% RSLogix 500 project LAB3_BW_OJ_BAK001.RSS, saved by version 8.40.00.08 %
PROJECT "UNTITLED"    % processor: MicroLogix 1400 %

PROGRAM FILES
  LAD 2   6 rungs

DATA FILES
  O0 OUTPUT  6 elements
  I1 INPUT  8 elements
  S2 STATUS  66 elements
  B3 BINARY  1 elements
  T4 TIMER  1 elements
  C5 COUNTER  1 elements
  R6 CONTROL  1 elements
  N7 INTEGER  1 elements
  F8 FLOAT  1 elements

LADDER 2
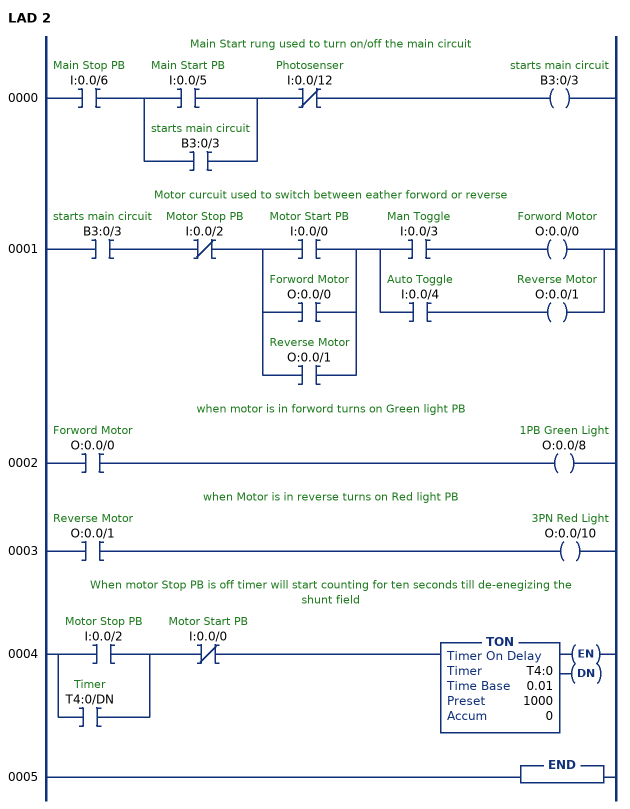
% Rung: 0 %
% Main Start rung used to turn on/off the main circuit %
SOR XIC I:0.0/6 BST XIC I:0.0/5 NXB XIC B3:0/3 BND XIO I:0.0/12 OTE B3:0/3 EOR
%   I:0.0/6  "Main Stop PB" %
%   I:0.0/5  "Main Start PB" %
%   B3:0/3  "starts main circuit" %
%   I:0.0/12  "Photosenser" %
% Rung: 1 %
% Motor curcuit used to switch between eather forword or reverse %
SOR XIC B3:0/3 XIO I:0.0/2 BST XIC I:0.0/0 NXB XIC O:0.0/0 NXB XIC O:0.0/1 BND BST XIC I:0.0/3 OTE O:0.0/0 NXB XIC I:0.0/4 OTE O:0.0/1 BND EOR
%   B3:0/3  "starts main circuit" %
%   I:0.0/2  "Motor Stop PB" %
%   I:0.0/0  "Motor Start PB" %
%   O:0.0/0  "Forword Motor" %
%   O:0.0/1  "Reverse Motor" %
%   I:0.0/3  "Man Toggle" %
%   I:0.0/4  "Auto Toggle" %
% Rung: 2 %
% when motor is in forword turns on Green light PB %
SOR XIC O:0.0/0 OTE O:0.0/8 EOR
%   O:0.0/0  "Forword Motor" %
%   O:0.0/8  "1PB Green Light" %
% Rung: 3 %
% when Motor is in reverse turns on Red light PB %
SOR XIC O:0.0/1 OTE O:0.0/10 EOR
%   O:0.0/1  "Reverse Motor" %
%   O:0.0/10  "3PN Red Light" %
% Rung: 4 %
% When motor Stop PB is off timer will start counting for ten seconds till de-enegizing the shunt field %
SOR BST XIC I:0.0/2 NXB XIC T4:0/DN BND XIO I:0.0/0 TON T4:0 0.01 1000 0 EOR
%   I:0.0/2  "Motor Stop PB" %
%   T4:0/DN  "Timer" %
%   I:0.0/0  "Motor Start PB" %
% Rung: 5 %
SOR END EOR

DATA TABLE (non-zero values as saved)
DATA T4
% .PRE .ACC %
% T4:0 % 1000 0
